{attribute addProperty BoxType "EL3356-0030-0025"}
{attribute addProperty Id "CtrlAT %Q*Ctrl_9754573E162"}
{attribute addProperty CRC "3563644232"}
{attribute addProperty SizeInBites "16"}
{attribute addProperty SizeInBytes "2"}
TYPE RMB_Control_D468E548 :
STRUCT
	{attribute addProperty Name "Ctrl"}
	Ctrl AT %Q* : Ctrl_9754573E;
END_STRUCT
END_TYPE

(* stored: Version 1.2.0.0, ProductVersion 3.1.4024.9
   DUT RMB_Control_D468E548: Id {e121892a-77d5-4403-b8ba-20d539c9a761} *)
